// TIA Portal V18 export
DATA_BLOCK "ZAxis_RelativeMotion_Test_DB"   // DB96
VERSION : 0.1
// stored: AutoNumber true, DBAccessibleFromOPCUA true, InstanceOfName ZAxis_RelativeMotion_Test, InstanceOfType FB
"ZAxis_RelativeMotion_Test"
   // VAR_INPUT
   //    StartTest : Bool;
   //    EndTest : Bool;
   //    AmountOfSteps : DInt;
   //    StepSizeInput : DInt;
   //    Position : DInt;
   //    AxisMoving : Bool;
   // END_VAR
   // VAR_OUTPUT
   //    StartTask : Bool;
   //    StepSize : DInt;
   //    StepNumber : DInt;
   //    CreateLogFile : Bool;
   //    StartLog : Bool;
   //    Comment : String;
   // END_VAR
   // VAR
   //    TestActiveInternal : Bool;
   //    ActualStep : DInt;
   //    StepCountNext : DInt;
   //    MovingInternal : Bool;
   //    ChangingCount : Bool;
   //    StartTaskM : Bool;
   //    LogCreatingReady : Bool;
   // END_VAR
BEGIN
END_DATA_BLOCK
